//A series of methods for use when testing functionality.
FUNCTION_BLOCK PUBLIC FB_Assert

METHOD FinishedTestingMsg
F_LogInfo('... Finished Testing');
END_METHOD

METHOD FINAL FloatsAreDifferent : BOOL
VAR_INPUT
	Float_1 : LREAL;
	Float_2 : LREAL;
	Precision : LREAL; // floating point precision.
	FailMsg : T_MaxString;
END_VAR
IF ABS(Float_1 - Float_2) <= Precision THEN
	F_LogError( 
		CONCAT('Assert.FloatsAreDifferent failed: ', FailMsg ) 
	);
ELSE
	FloatsAreDifferent := TRUE;
END_IF
END_METHOD

METHOD FINAL FloatsAreEqual : BOOL
VAR_INPUT
	Float_1 : LREAL;
	Float_2 : LREAL;
	Precision : LREAL; // floating point precision.
	FailMsg : T_MaxString;
END_VAR
IF ABS(Float_1 - Float_2) > Precision THEN
	F_LogError( 
		CONCAT('Assert.FloatsAreEqual failed: ', FailMsg ) 
	);
ELSE
	FloatsAreEqual := TRUE;
END_IF
END_METHOD

METHOD FINAL IsFalse : BOOL
VAR_INPUT
	Condition : BOOL;
	FailMsg : T_MaxString;
END_VAR
IF Condition THEN
	F_LogError( 
		CONCAT( 'Assert.IsFalse failed: ', FailMsg ) 
	);	
ELSE
	IsFalse := TRUE;
END_IF
END_METHOD

METHOD FINAL IsTrue : BOOL
VAR_INPUT
	Condition : BOOL;
	FailMsg : T_MaxString;
END_VAR
IF NOT Condition THEN
	F_LogError( 
		CONCAT( 'Assert.IsTrue failed: ', FailMsg ) 
	);
ELSE
	IsTrue := TRUE;
END_IF
END_METHOD

METHOD PUBLIC StartTestingMsg
F_LogInfo('Testing started...');
END_METHOD

END_FUNCTION_BLOCK

(* stored: Version 1.1.0.1, ProductVersion 3.1.4020.12
   POU FB_Assert: Id {ecb56ce5-5949-45d6-a7a3-6a44bf4e9be1}, SpecialFunc None
   Method FinishedTestingMsg: Id {106987b1-ce00-47e4-aac5-d476825cced6}
   Method FloatsAreDifferent: Id {ab1883dd-fa0d-4b4f-ab8d-1b1323d1918b}
   Method FloatsAreEqual: Id {77593574-aaba-4f16-88d4-b5011110ee23}
   Method IsFalse: Id {93a463f2-4d73-4cc3-b90b-0a8fb8b299f2}
   Method IsTrue: Id {f4a50788-6073-4164-9cb5-a901d67a227a}
   Method StartTestingMsg: Id {01264389-f134-4d34-bb86-b5a5b91ced6b} *)
